    tonConveyorLevelerHomingTimeout(IN := FALSE);
    tonConveyorLevelerBrakeReleaseDelay(IN := FALSE);
    tonConveyorLevelerBrakeHoldDelay(IN := FALSE);

    conveyorLevelerFault := TRUE;
    conveyorLevelerFaultCode := 2;
    conveyorLevelerControlState := E_ConveyorLevelerState.FAULT;


ELSIF NOT conveyorLevelerDriveOk THEN

    conveyorLevelerState := 'DRIVE_NOT_OK';

    tonConveyorLevelerHomingTimeout(IN := FALSE);
    tonConveyorLevelerBrakeReleaseDelay(IN := FALSE);
    tonConveyorLevelerBrakeHoldDelay(IN := FALSE);

    conveyorLevelerFault := TRUE;
    conveyorLevelerFaultCode := 1;
    conveyorLevelerControlState := E_ConveyorLevelerState.FAULT;


ELSIF conveyorLevelerUpperSafetyLimit THEN

    conveyorLevelerState := 'UPPER_SAFE_LIMIT';

    tonConveyorLevelerHomingTimeout(IN := FALSE);
    tonConveyorLevelerBrakeReleaseDelay(IN := FALSE);
    tonConveyorLevelerBrakeHoldDelay(IN := FALSE);

    conveyorLevelerFault := TRUE;
    conveyorLevelerFaultCode := 4;
    conveyorLevelerControlState := E_ConveyorLevelerState.FAULT;


ELSIF conveyorLevelerLowerSafetyLimit THEN

    conveyorLevelerState := 'LOWER_SAFE_LIMIT';

    tonConveyorLevelerHomingTimeout(IN := FALSE);
    tonConveyorLevelerBrakeReleaseDelay(IN := FALSE);
    tonConveyorLevelerBrakeHoldDelay(IN := FALSE);

    conveyorLevelerFault := TRUE;
    conveyorLevelerFaultCode := 5;
    conveyorLevelerControlState := E_ConveyorLevelerState.FAULT;


ELSIF NOT systemRunEnable THEN

    // EN: Master stop disables movement without generating an axis fault.
    conveyorLevelerState := 'SYSTEM_DISABLED';

    conveyorLevelerSignedSpeedRefMmps := 0.0;

    tonConveyorLevelerHomingTimeout(IN := FALSE);
    tonConveyorLevelerBrakeReleaseDelay(IN := FALSE);
    tonConveyorLevelerBrakeHoldDelay(IN := FALSE);

    IF conveyorLevelerControlState <> E_ConveyorLevelerState.FAULT THEN
        conveyorLevelerControlState := E_ConveyorLevelerState.STOP;
    END_IF


ELSE

    //==============================================================
    // 9) Mode selection
    //==============================================================
    // EN: Homing has priority over manual and automatic leveling.
    IF rConveyorLevelerHome AND NOT conveyorLevelerFault THEN
        conveyorLevelerControlState := E_ConveyorLevelerState.HOME_FAST_SEARCH;
    END_IF;


    //==============================================================
    // 10) Conveyor leveler state machine
    //==============================================================
    CASE conveyorLevelerControlState OF

        E_ConveyorLevelerState.STOP: // STOP
            conveyorLevelerState := 'STOP';

            tonConveyorLevelerHomingTimeout(IN := FALSE);

            IF conveyorLevelerUpCmd OR conveyorLevelerDownCmd THEN

                conveyorLevelerControlState := E_ConveyorLevelerState.MANUAL;

            ELSIF conveyorLevelerAutoCmd THEN

                conveyorLevelerControlState := E_ConveyorLevelerState.AUTO_LEVELING;

            END_IF


        E_ConveyorLevelerState.HOME_FAST_SEARCH: // HOME_FAST_SEARCH
            conveyorLevelerState := 'HOME_FAST';

            conveyorLevelerHomed := FALSE;
            conveyorLevelerInPosition := FALSE;

            tonConveyorLevelerHomingTimeout(
                IN := TRUE,
                PT := machineConfig.conveyorLevelerHomingTimeout
            );

            IF tonConveyorLevelerHomingTimeout.Q THEN

                conveyorLevelerSignedSpeedRefMmps := 0.0;

                tonConveyorLevelerHomingTimeout(IN := FALSE);

                conveyorLevelerFault := TRUE;
                conveyorLevelerFaultCode := 3;

                conveyorLevelerState := 'HOME_TIMEOUT';
                conveyorLevelerControlState := E_ConveyorLevelerState.FAULT;


            ELSIF conveyorLevelerHomeLimitReached THEN

                // EN: Lower home sensor found. Stop and start slow exit.
                conveyorLevelerSignedSpeedRefMmps := 0.0;

                conveyorLevelerControlState := E_ConveyorLevelerState.HOME_SLOW_EXIT_SENSOR;


            ELSE

                IF conveyorLevelerHomeMoveAllowed THEN

                    // EN: Fast search moves down to find the lower home sensor.
                    conveyorLevelerSignedSpeedRefMmps :=
                        -ABS(machineConfig.conveyorLevelerHomingSpeedMmps);

                ELSE

                    conveyorLevelerSignedSpeedRefMmps := 0.0;

                END_IF

            END_IF


        E_ConveyorLevelerState.HOME_SLOW_EXIT_SENSOR: // HOME_SLOW_EXIT_SENSOR
            conveyorLevelerState := 'HOME_SLOW_EXIT';

            tonConveyorLevelerHomingTimeout(
                IN := TRUE,
                PT := machineConfig.conveyorLevelerHomingTimeout
            );

            IF tonConveyorLevelerHomingTimeout.Q THEN

                conveyorLevelerSignedSpeedRefMmps := 0.0;

                tonConveyorLevelerHomingTimeout(IN := FALSE);

                conveyorLevelerFault := TRUE;
                conveyorLevelerFaultCode := 3;

                conveyorLevelerState := 'HOME_TIMEOUT';
                conveyorLevelerControlState := E_ConveyorLevelerState.FAULT;


            ELSIF conveyorLevelerHomeLimitFallingEdge THEN

                // EN: Lower home sensor falling edge found.
                //     Stop before setting encoder.
                conveyorLevelerSignedSpeedRefMmps := 0.0;

                tonConveyorLevelerHomingTimeout(IN := FALSE);

                conveyorLevelerControlState := E_ConveyorLevelerState.HOME_SET_ENCODER;


            ELSE

                IF conveyorLevelerHomeMoveAllowed THEN

                    // EN: Slow exit moves up until leaving the lower home sensor.
                    conveyorLevelerSignedSpeedRefMmps :=
                        ABS(machineConfig.conveyorLevelerMinMoveSpeedMmps);

                ELSE

                    conveyorLevelerSignedSpeedRefMmps := 0.0;

                END_IF

            END_IF


        E_ConveyorLevelerState.HOME_SET_ENCODER: // HOME_SET_ENCODER
            conveyorLevelerState := 'HOME_SET_ENCODER';

            conveyorLevelerSignedSpeedRefMmps := 0.0;

            tonConveyorLevelerHomingTimeout(IN := FALSE);

            // EN: Set encoder only after leaving the home sensor edge.
            conveyorLevelerSetEncoderPositionTrigger := TRUE;
            conveyorLevelerSetEncoderPositionMm :=
                machineConfig.conveyorLevelerMinPositionMm;

            conveyorLevelerHomed := TRUE;
            conveyorLevelerFault := FALSE;
            conveyorLevelerFaultCode := 0;

            IF conveyorLevelerAutoCmd THEN
                conveyorLevelerControlState := E_ConveyorLevelerState.AUTO_LEVELING;
            ELSE
                conveyorLevelerControlState := E_ConveyorLevelerState.STOP;
            END_IF


        E_ConveyorLevelerState.MANUAL: // MANUAL
            conveyorLevelerState := 'MANUAL';

            tonConveyorLevelerHomingTimeout(IN := FALSE);

            IF conveyorLevelerUpCmd AND conveyorLevelerDownCmd THEN

                conveyorLevelerSignedSpeedRefMmps := 0.0;


            ELSIF conveyorLevelerUpCmd THEN

                IF conveyorLevelerUpAllowed THEN

                    conveyorLevelerSignedSpeedRefMmps :=
                        ABS(machineConfig.conveyorLevelerManualSpeedMmps);

                ELSE

                    conveyorLevelerSignedSpeedRefMmps := 0.0;

                END_IF


            ELSIF conveyorLevelerDownCmd THEN

                IF conveyorLevelerDownAllowed THEN

                    conveyorLevelerSignedSpeedRefMmps :=
                        -ABS(machineConfig.conveyorLevelerManualSpeedMmps);

                ELSE

                    conveyorLevelerSignedSpeedRefMmps := 0.0;

                END_IF


            ELSE

                conveyorLevelerSignedSpeedRefMmps := 0.0;

                IF conveyorLevelerAutoCmd THEN

                    conveyorLevelerControlState := E_ConveyorLevelerState.AUTO_LEVELING;

                ELSE

                    conveyorLevelerControlState := E_ConveyorLevelerState.STOP;

                END_IF

            END_IF


        E_ConveyorLevelerState.AUTO_LEVELING: // AUTO_LEVELING
            conveyorLevelerState := 'AUTO_LEVELING';

            tonConveyorLevelerHomingTimeout(IN := FALSE);

            IF NOT conveyorLevelerAutoCmd THEN

                conveyorLevelerSignedSpeedRefMmps := 0.0;
                conveyorLevelerControlState := E_ConveyorLevelerState.STOP;


            ELSIF NOT conveyorLevelerHomed THEN

                // EN: Automatic leveling is blocked before homing.
                conveyorLevelerSignedSpeedRefMmps := 0.0;
                conveyorLevelerState := 'AUTO_NO_HOME';


            ELSIF conveyorLevelerInPosition THEN

                conveyorLevelerSignedSpeedRefMmps := 0.0;


            ELSE

                // EN: Simple proportional position control.
                conveyorLevelerRawSpeedRefMmps :=
                    conveyorLevelerPositionErrorMm *
                    machineConfig.conveyorLevelerPositionKp;

                conveyorLevelerRawSpeedRefMmps :=
                    LIMIT(
                        -ABS(machineConfig.conveyorLevelerAutoMaxSpeedMmps),
                        conveyorLevelerRawSpeedRefMmps,
                        ABS(machineConfig.conveyorLevelerAutoMaxSpeedMmps)
                    );

                // EN: Apply minimum movement speed to overcome friction.
                IF ABS(conveyorLevelerRawSpeedRefMmps) <
                   ABS(machineConfig.conveyorLevelerMinMoveSpeedMmps) THEN

                    IF conveyorLevelerPositionErrorMm > 0.0 THEN

                        conveyorLevelerRawSpeedRefMmps :=
                            ABS(machineConfig.conveyorLevelerMinMoveSpeedMmps);

                    ELSE

                        conveyorLevelerRawSpeedRefMmps :=
                            -ABS(machineConfig.conveyorLevelerMinMoveSpeedMmps);

                    END_IF

                END_IF

                // EN: Apply limit protection according to movement direction.
                IF (conveyorLevelerRawSpeedRefMmps > 0.0) AND conveyorLevelerUpAllowed THEN

                    conveyorLevelerSignedSpeedRefMmps := conveyorLevelerRawSpeedRefMmps;

                ELSIF (conveyorLevelerRawSpeedRefMmps < 0.0) AND conveyorLevelerDownAllowed THEN

                    conveyorLevelerSignedSpeedRefMmps := conveyorLevelerRawSpeedRefMmps;

                ELSE

                    conveyorLevelerSignedSpeedRefMmps := 0.0;

                END_IF

            END_IF


        E_ConveyorLevelerState.FAULT: // FAULT
            conveyorLevelerState := 'FAULT';

            conveyorLevelerSignedSpeedRefMmps := 0.0;

            tonConveyorLevelerHomingTimeout(IN := FALSE);

            IF resetCmd AND
               safetyCircuitOk AND
               conveyorLevelerDriveOk AND
               NOT conveyorLevelerUpperSafetyLimit AND
               NOT conveyorLevelerLowerSafetyLimit THEN

                conveyorLevelerFault := FALSE;
                conveyorLevelerFaultCode := 0;
                conveyorLevelerControlState := E_ConveyorLevelerState.STOP;

            END_IF


    ELSE

        conveyorLevelerControlState := E_ConveyorLevelerState.STOP;

    END_CASE;

END_IF;


//==============================================================
// 11) Encoder set pulse
//==============================================================
// EN: Extend encoder set command to ensure the encoder block sees it.
tpConveyorLevelerSetEncoderPosition(
    IN := conveyorLevelerSetEncoderPositionTrigger,
    PT := machineConfig.conveyorLevelerSetEncoderPulseTime
);

conveyorLevelerSetEncoderPosition := tpConveyorLevelerSetEncoderPosition.Q;


//==============================================================
// 12) Brake release control
//==============================================================
// EN: A movement request keeps the magnetic brake released.
//     After movement stops, the brake remains released for a hold time.
conveyorLevelerMoveRequest :=
    systemRunEnable AND
    safetyCircuitOk AND
    conveyorLevelerDriveOk AND
    NOT conveyorLevelerFault AND
    (ABS(conveyorLevelerSignedSpeedRefMmps) >= machineConfig.conveyorLevelerRunMinSpeedMmps);


IF conveyorLevelerMoveRequest THEN

    conveyorLevelerBrakeReleaseRequest := TRUE;

    tonConveyorLevelerBrakeHoldDelay(IN := FALSE);

ELSE

    IF conveyorLevelerBrakeRelease THEN

        tonConveyorLevelerBrakeHoldDelay(
            IN := TRUE,
            PT := machineConfig.conveyorLevelerBrakeHoldTime
        );

        conveyorLevelerBrakeReleaseRequest :=
            NOT tonConveyorLevelerBrakeHoldDelay.Q;

    ELSE

        tonConveyorLevelerBrakeHoldDelay(IN := FALSE);
        conveyorLevelerBrakeReleaseRequest := FALSE;

    END_IF

END_IF;


conveyorLevelerBrakeRelease :=
    systemRunEnable AND
    safetyCircuitOk AND
    conveyorLevelerDriveOk AND
    NOT conveyorLevelerFault AND
    conveyorLevelerBrakeReleaseRequest;


//==============================================================
// 13) Brake release delay before motor movement
//==============================================================
// EN: The motor can run only after brake release delay.
tonConveyorLevelerBrakeReleaseDelay(
    IN := conveyorLevelerMoveRequest AND conveyorLevelerBrakeRelease,
    PT := machineConfig.conveyorLevelerBrakeReleaseDelay
);


//==============================================================
// 14) Conveyor leveler direction and speed outputs
//==============================================================
// EN: Convert signed internal speed command into direction outputs
//     and positive speed reference.
IF conveyorLevelerMoveRequest AND
   conveyorLevelerBrakeRelease AND
   tonConveyorLevelerBrakeReleaseDelay.Q THEN

    conveyorLevelerSpeedRefMmps :=
        ABS(conveyorLevelerSignedSpeedRefMmps);

    conveyorLevelerRunUp :=
        conveyorLevelerSignedSpeedRefMmps > 0.0;

    conveyorLevelerRunDown :=
        conveyorLevelerSignedSpeedRefMmps < 0.0;

ELSE

    conveyorLevelerSpeedRefMmps := 0.0;

    conveyorLevelerRunUp := FALSE;
    conveyorLevelerRunDown := FALSE;

END_IF;
END_METHOD

//==============================================================
// SIMPLE STACKER — SPEED REFERENCE GENERATOR
// EN: Generates synchronized and sheet-stack separation speed references [m/min].
//==============================================================
METHOD _ConveyorSpeedControl
VAR
packageGapReady                   : BOOL;
    validCycleTimeS                   : REAL;

    sheetConveyorsSpeedUpReferenceMPM : REAL;

    sheetConveyor1BaseSpeedMPM        : REAL;
    sheetConveyor2BaseSpeedMPM        : REAL;
    sheetConveyor3BaseSpeedMPM        : REAL;
END_VAR


//==============================================================
// 1) Default event pulses
//==============================================================
sheetStackSeparationStarted         := FALSE;
sheetStackSeparationFinished        := FALSE;

sheetConveyor2SeparationStarted     := FALSE;
sheetConveyor2SeparationFinished    := FALSE;

sheetConveyor3SeparationStarted     := FALSE;
sheetConveyor3SeparationFinished    := FALSE;


//==============================================================
// 2) Enable and scan time
//==============================================================
speedControlEnabled :=
    sheetConveyor1Run AND
    sheetConveyor2Run AND
    sheetConveyor3Run AND
    safetyCircuitOk;

rampReset := NOT speedControlEnabled;


// EN: Read PLC scan time using OSCAT CYCLE_TIME.
instCycleTime(
    RST := resetCmd
);


// EN: Convert last cycle time from TIME/ms to seconds.
scanTimeMs := TIME_TO_REAL(instCycleTime.ct_last);

validCycleTimeS :=
    LIMIT(
        0.001,
        scanTimeMs / 1000.0,
        20.0
    );

scanTimeS := validCycleTimeS;



//==============================================================
// 4) Calculate normal stacker speed
//==============================================================
IF speedControlEnabled THEN

    normalStackerSpeedMPM :=
        LIMIT(
            machineConfig.minimumSpeedMPM,
            MAX(0.0, lineSpeedMPM) *
                MAX(0.0, machineConfig.stackerSpeedRatio),
            machineConfig.maximumSpeedMPM
        );

ELSE

    normalStackerSpeedMPM := 0.0;

END_IF;


//==============================================================
// 6) Calculate normal speed for each conveyor
//==============================================================
sheetConveyor1NormalSpeedMPM :=
    normalStackerSpeedMPM *
    MAX(0.0, machineConfig.sheetConveyor1SpeedTrim);

sheetConveyor2NormalSpeedMPM :=
    normalStackerSpeedMPM *
    MAX(0.0, machineConfig.sheetConveyor2SpeedTrim);

sheetConveyor3NormalSpeedMPM :=
    normalStackerSpeedMPM *
    MAX(0.0, machineConfig.sheetConveyor3SpeedTrim);


//==============================================================
// 6.1) Sheet conveyors speed-up reference
//==============================================================
// EN: Speed-up is added directly to conveyors 1/2/3 references.
//     It can work even when line speed is zero, as long as the
//     conveyor group is enabled.
IF speedControlEnabled AND sheetConveyorsSpeedUpCmd THEN

    sheetConveyorsSpeedUpReferenceMPM :=
        MAX(0.0, machineConfig.sheetConveyorsSpeedUpMPM);

ELSE

    sheetConveyorsSpeedUpReferenceMPM := 0.0;

END_IF;


//==============================================================
// 6.2) Base speed references including speed-up
//==============================================================
// EN: Base speed is the synchronized conveyor speed plus operator speed-up.
//     Separation tracking must use this base speed as reference.
sheetConveyor1BaseSpeedMPM :=
    sheetConveyor1NormalSpeedMPM + sheetConveyorsSpeedUpReferenceMPM;

sheetConveyor2BaseSpeedMPM :=
    sheetConveyor2NormalSpeedMPM + sheetConveyorsSpeedUpReferenceMPM;

sheetConveyor3BaseSpeedMPM :=
    sheetConveyor3NormalSpeedMPM + sheetConveyorsSpeedUpReferenceMPM;


//==============================================================
// 7) Calculate separation high speed
//==============================================================
// EN: Gap speed also receives the same speed-up reference.
//     This preserves the real gap differential while allowing operator boost.
sheetConveyor2GapSpeedMPM :=
    (sheetConveyor2NormalSpeedMPM * MAX(0.0, machineConfig.packageGapSpeedRatio)) +
    machineConfig.packageGapSpeedOffsetMPM +
    sheetConveyorsSpeedUpReferenceMPM;

sheetConveyor3GapSpeedMPM :=
    (sheetConveyor3NormalSpeedMPM * MAX(0.0, machineConfig.packageGapSpeedRatio)) +
    machineConfig.packageGapSpeedOffsetMPM +
    sheetConveyorsSpeedUpReferenceMPM;


//==============================================================
// 8) Calculate separation tracking target distances
//==============================================================
// EN: Separation tracking target is based on each conveyor length.
sheetConveyor2TargetDistanceM :=
    MAX(0.0, machineConfig.sheetConveyor2LengthM);

sheetConveyor3TargetDistanceM :=
    MAX(0.0, machineConfig.sheetConveyor3LengthM);


//==============================================================
// 9) Check separation ready conditions
//==============================================================
// EN: Compare gap speed against base speed, not normal speed.
//     Otherwise operator speed-up would be incorrectly counted as gap opening.
packageGapReady :=
    speedControlEnabled AND
    (sheetConveyor2TargetDistanceM > 0.0) AND
    (sheetConveyor3TargetDistanceM > 0.0) AND
    ((sheetConveyor2GapSpeedMPM - sheetConveyor2BaseSpeedMPM) >= machineConfig.minimumOpeningSpeedMPM) AND
    ((sheetConveyor3GapSpeedMPM - sheetConveyor3BaseSpeedMPM) >= machineConfig.minimumOpeningSpeedMPM);

sheetStackSeparationReady := packageGapReady;


//==============================================================
// 9) Sheet stack separation state machine
//==============================================================
IF NOT speedControlEnabled THEN

    sheetStackSeparationState      := 'DISABLED';
    sheetStackSeparationStateCode  := -1;

    packageSeparationState         := E_PackageSeparationState.NORMAL;

    sheetStackSeparationActive     := FALSE;
    sheetStackBrakeActive          := FALSE;
    brakeValve                     := FALSE;

    sheetConveyor2SeparationActive := FALSE;
    sheetConveyor3SeparationActive := FALSE;

    sheetConveyor2HighSpeedActive  := FALSE;
    sheetConveyor3HighSpeedActive  := FALSE;

    sheetConveyor2OpeningDistanceM := 0.0;
    sheetConveyor3OpeningDistanceM := 0.0;

    sheetConveyor1TargetSpeedMPM   := 0.0;
    sheetConveyor2TargetSpeedMPM   := 0.0;
    sheetConveyor3TargetSpeedMPM   := 0.0;


ELSE

    CASE packageSeparationState OF

        E_PackageSeparationState.NORMAL: // NORMAL
            sheetStackSeparationState     := 'NORMAL';
            sheetStackSeparationStateCode := 0;

            sheetStackSeparationActive    := FALSE;
            sheetStackBrakeActive         := FALSE;
            brakeValve                    := FALSE;

            sheetConveyor2SeparationActive := FALSE;
            sheetConveyor3SeparationActive := FALSE;

            sheetConveyor2HighSpeedActive  := FALSE;
            sheetConveyor3HighSpeedActive  := FALSE;

            sheetConveyor2OpeningDistanceM := 0.0;
            sheetConveyor3OpeningDistanceM := 0.0;

            sheetConveyor1TargetSpeedMPM  := sheetConveyor1BaseSpeedMPM;
            sheetConveyor2TargetSpeedMPM  := sheetConveyor2BaseSpeedMPM;
            sheetConveyor3TargetSpeedMPM  := sheetConveyor3BaseSpeedMPM;

            IF rPackageComplete AND packageGapReady THEN
                packageSeparationState := E_PackageSeparationState.START_SEPARATION;
            END_IF


        E_PackageSeparationState.START_SEPARATION: // START_SHEET_STACK_SEPARATION
            sheetStackSeparationState     := 'START_SEPARATION';
            sheetStackSeparationStateCode := 10;

            sheetStackSeparationActive    := TRUE;
            sheetStackSeparationStarted   := TRUE;

            sheetStackBrakeActive         := TRUE;
            brakeValve                    := TRUE;

            // EN: Conveyor 2 tracking starts immediately.
            sheetConveyor2SeparationStarted := TRUE;

            sheetConveyor2SeparationActive  := TRUE;
            sheetConveyor3SeparationActive  := FALSE;

            // EN: Conveyor 2 and 3 accelerate together from the beginning.
            sheetConveyor2HighSpeedActive   := TRUE;
            sheetConveyor3HighSpeedActive   := TRUE;

            sheetConveyor2OpeningDistanceM  := 0.0;
            sheetConveyor3OpeningDistanceM  := 0.0;

            sheetConveyor1TargetSpeedMPM    := sheetConveyor1BaseSpeedMPM;
            sheetConveyor2TargetSpeedMPM    := sheetConveyor2GapSpeedMPM;
            sheetConveyor3TargetSpeedMPM    := sheetConveyor3GapSpeedMPM;

            packageSeparationState := E_PackageSeparationState.CONVEYOR_2_TRACKING;


        E_PackageSeparationState.CONVEYOR_2_TRACKING: // SHEET_CONVEYOR_2_SEPARATION_TRACKING
            sheetStackSeparationState     := 'CONV2_TRACKING';
            sheetStackSeparationStateCode := 20;

            sheetStackSeparationActive    := TRUE;

            sheetStackBrakeActive         := TRUE;
            brakeValve                    := TRUE;

            sheetConveyor2SeparationActive := TRUE;
            sheetConveyor3SeparationActive := FALSE;

            sheetConveyor2HighSpeedActive  := TRUE;
            sheetConveyor3HighSpeedActive  := TRUE;

            sheetConveyor1TargetSpeedMPM  := sheetConveyor1BaseSpeedMPM;
            sheetConveyor2TargetSpeedMPM  := sheetConveyor2GapSpeedMPM;
            sheetConveyor3TargetSpeedMPM  := sheetConveyor3GapSpeedMPM;

            IF sheetConveyor2OpeningDistanceM >= sheetConveyor2TargetDistanceM THEN

                // EN: Conveyor 2 tracking finished. Conveyor 2 returns to base speed.
                sheetConveyor2SeparationFinished := TRUE;

                sheetConveyor2SeparationActive   := FALSE;
                sheetConveyor2HighSpeedActive    := FALSE;

                sheetStackBrakeActive            := FALSE;
                brakeValve                       := FALSE;

                sheetConveyor2TargetSpeedMPM     := sheetConveyor2BaseSpeedMPM;

                // EN: Conveyor 3 tracking starts after conveyor 2 returns to sync.
                sheetConveyor3SeparationStarted := TRUE;
                sheetConveyor3OpeningDistanceM  := 0.0;

                packageSeparationState := E_PackageSeparationState.CONVEYOR_3_TRACKING;

            END_IF


        E_PackageSeparationState.CONVEYOR_3_TRACKING: // SHEET_CONVEYOR_3_SEPARATION_TRACKING
            sheetStackSeparationState     := 'CONV3_TRACKING';
            sheetStackSeparationStateCode := 30;

            sheetStackSeparationActive    := TRUE;

            sheetStackBrakeActive         := FALSE;
            brakeValve                    := FALSE;

            sheetConveyor2SeparationActive := FALSE;
            sheetConveyor3SeparationActive := TRUE;

            sheetConveyor2HighSpeedActive  := FALSE;
            sheetConveyor3HighSpeedActive  := TRUE;

            sheetConveyor1TargetSpeedMPM  := sheetConveyor1BaseSpeedMPM;
            sheetConveyor2TargetSpeedMPM  := sheetConveyor2BaseSpeedMPM;
            sheetConveyor3TargetSpeedMPM  := sheetConveyor3GapSpeedMPM;

            IF sheetConveyor3OpeningDistanceM >= sheetConveyor3TargetDistanceM THEN

                // EN: Conveyor 3 returns to base synchronized speed.
                sheetConveyor3TargetSpeedMPM := sheetConveyor3BaseSpeedMPM;

                packageSeparationState := E_PackageSeparationState.FINISH_SEPARATION;

            END_IF


        E_PackageSeparationState.FINISH_SEPARATION: // FINISH_SHEET_STACK_SEPARATION
            sheetStackSeparationState     := 'FINISH_SEPARATION';
            sheetStackSeparationStateCode := 40;

            sheetStackSeparationActive    := FALSE;
            sheetStackSeparationFinished  := TRUE;

            sheetStackBrakeActive         := FALSE;
            brakeValve                    := FALSE;

            sheetConveyor2SeparationActive  := FALSE;
            sheetConveyor3SeparationActive  := FALSE;

            sheetConveyor2HighSpeedActive   := FALSE;
            sheetConveyor3HighSpeedActive   := FALSE;

            sheetConveyor3SeparationFinished := TRUE;

            sheetConveyor1TargetSpeedMPM  := sheetConveyor1BaseSpeedMPM;
            sheetConveyor2TargetSpeedMPM  := sheetConveyor2BaseSpeedMPM;
            sheetConveyor3TargetSpeedMPM  := sheetConveyor3BaseSpeedMPM;

            packageSeparationState := E_PackageSeparationState.NORMAL;


    ELSE

        packageSeparationState := E_PackageSeparationState.NORMAL;

    END_CASE;

END_IF;


//==============================================================
// 10) Limit speed targets
//==============================================================
sheetConveyor1TargetSpeedMPM := LIMIT(
    machineConfig.minimumSpeedMPM,
    sheetConveyor1TargetSpeedMPM,
    machineConfig.maximumSpeedMPM
);

sheetConveyor2TargetSpeedMPM := LIMIT(
    machineConfig.minimumSpeedMPM,
    sheetConveyor2TargetSpeedMPM,
    machineConfig.maximumSpeedMPM
);

sheetConveyor3TargetSpeedMPM := LIMIT(
    machineConfig.minimumSpeedMPM,
    sheetConveyor3TargetSpeedMPM,
    machineConfig.maximumSpeedMPM
);


//==============================================================
// 12) Ramp sheet conveyor 1 speed reference
//==============================================================
instRampSheetConveyor1(
    X          := sheetConveyor1TargetSpeedMPM,
    A_UP       := MAX(0.0, machineConfig.rampAccelerationUpMPMps2),
    A_DN       := -MAX(0.0, machineConfig.rampAccelerationDownMPMps2),
    VU_MAX     := MAX(0.0, machineConfig.rampVelocityUpMaxMPMps),
    VD_MAX     := -MAX(0.0, machineConfig.rampVelocityDownMaxMPMps),
    LIMIT_HIGH := machineConfig.maximumSpeedMPM,
    LIMIT_LOW  := machineConfig.minimumSpeedMPM,
    RST        := rampReset,
    Y          => sheetConveyor1SpeedRefMPM
);


//==============================================================
// 13) Ramp sheet conveyor 2 speed reference
//==============================================================
instRampSheetConveyor2(
    X          := sheetConveyor2TargetSpeedMPM,
    A_UP       := MAX(0.0, machineConfig.rampAccelerationUpMPMps2),
    A_DN       := -MAX(0.0, machineConfig.rampAccelerationDownMPMps2),
    VU_MAX     := MAX(0.0, machineConfig.rampVelocityUpMaxMPMps),
    VD_MAX     := -MAX(0.0, machineConfig.rampVelocityDownMaxMPMps),
    LIMIT_HIGH := machineConfig.maximumSpeedMPM,
    LIMIT_LOW  := machineConfig.minimumSpeedMPM,
    RST        := rampReset,
    Y          => sheetConveyor2SpeedRefMPM
);


//==============================================================
// 14) Ramp sheet conveyor 3 speed reference
//==============================================================
instRampSheetConveyor3(
    X          := sheetConveyor3TargetSpeedMPM,
    A_UP       := MAX(0.0, machineConfig.rampAccelerationUpMPMps2),
    A_DN       := -MAX(0.0, machineConfig.rampAccelerationDownMPMps2),
    VU_MAX     := MAX(0.0, machineConfig.rampVelocityUpMaxMPMps),
    VD_MAX     := -MAX(0.0, machineConfig.rampVelocityDownMaxMPMps),
    LIMIT_HIGH := machineConfig.maximumSpeedMPM,
    LIMIT_LOW  := machineConfig.minimumSpeedMPM,
    RST        := rampReset,
    Y          => sheetConveyor3SpeedRefMPM
);


//==============================================================
// 16) Calculate real separation tracking speed using ramped references
//==============================================================
// EN: Only the real speed differential above the base speed moves the
//     separation point through the conveyors.
//     Operator speed-up is already included in base speed, so it is not
//     counted as gap opening.
sheetConveyor2OpeningSpeedMPM :=
    MAX(0.0, sheetConveyor2SpeedRefMPM - sheetConveyor2BaseSpeedMPM);

sheetConveyor3OpeningSpeedMPM :=
    MAX(0.0, sheetConveyor3SpeedRefMPM - sheetConveyor3BaseSpeedMPM);


//==============================================================
// 17) Integrate real separation tracking distance
//==============================================================
IF speedControlEnabled THEN

    IF packageSeparationState = E_PackageSeparationState.CONVEYOR_2_TRACKING THEN

        IF sheetConveyor2OpeningSpeedMPM >= machineConfig.minimumOpeningSpeedMPM THEN

            sheetConveyor2OpeningDistanceM :=
                sheetConveyor2OpeningDistanceM +
                (sheetConveyor2OpeningSpeedMPM / 60.0) * scanTimeS;

        END_IF

    ELSIF packageSeparationState = E_PackageSeparationState.CONVEYOR_3_TRACKING THEN

        IF sheetConveyor3OpeningSpeedMPM >= machineConfig.minimumOpeningSpeedMPM THEN

            sheetConveyor3OpeningDistanceM :=
                sheetConveyor3OpeningDistanceM +
                (sheetConveyor3OpeningSpeedMPM / 60.0) * scanTimeS;

        END_IF

    END_IF

END_IF;


//==============================================================
// 18) Publish tracking distances to outputs
//==============================================================
sheetConveyor2TrackingDistanceM := sheetConveyor2OpeningDistanceM;
sheetConveyor3TrackingDistanceM := sheetConveyor3OpeningDistanceM;
END_METHOD

//==============================================================
// SIMPLE STACKER — HMI STATUS
// EN: Maps internal status, outputs, positions and diagnostics
//     to the HMI status structure.
//==============================================================
METHOD _HmiStatus



//==============================================================
// 1) System general status
//==============================================================
hmiStatus.systemRunEnable :=
    systemRunEnable;

hmiStatus.safetyCircuitOk :=
    safetyCircuitOk;

hmiStatus.faultActive :=
    faultActive OR
    backstopFault OR
    conveyorLevelerFault OR
    sheetStackDischargeFault OR
    sheetStackDischargeConveyorFault;

hmiStatus.deviceState :=
    deviceState;


//==============================================================
// 2) Sheet conveyor group status
//==============================================================
hmiStatus.synchronizedConveyorsRunning :=
    synchronizedConveyorsRunning;

hmiStatus.sheetConveyor1Run :=
    sheetConveyor1Run;

hmiStatus.sheetConveyor2Run :=
    sheetConveyor2Run;

hmiStatus.sheetConveyor3Run :=
    sheetConveyor3Run;

hmiStatus.sheetConveyor1SpeedRefMPM :=
    sheetConveyor1SpeedRefMPM;

hmiStatus.sheetConveyor2SpeedRefMPM :=
    sheetConveyor2SpeedRefMPM;

hmiStatus.sheetConveyor3SpeedRefMPM :=
    sheetConveyor3SpeedRefMPM;

CASE syncConveyorsState OF
    E_SyncConveyorsState.IDLE:
        hmiStatus.syncConveyorsState := 0;

    E_SyncConveyorsState.RUN:
        hmiStatus.syncConveyorsState := 1;

    E_SyncConveyorsState.FAULT:
        hmiStatus.syncConveyorsState := 10;

ELSE
    hmiStatus.syncConveyorsState := 0;
END_CASE;


//==============================================================
// 3) Sheet stack separation status
//==============================================================
hmiStatus.sheetStackSeparationReady :=
    sheetStackSeparationReady;

hmiStatus.sheetStackSeparationActive :=
    sheetStackSeparationActive;

hmiStatus.sheetStackBrakeActive :=
    sheetStackBrakeActive;


//==============================================================
// 4) Sheet stack discharge sequence status
//==============================================================
hmiStatus.sheetStackDischargeState :=
    sheetStackDischargeState;

hmiStatus.sheetStackDischargeStateCode :=
    sheetStackDischargeStateCode;

hmiStatus.sheetStackDischargePending :=
    sheetStackDischargePending;

hmiStatus.sheetStackDischargeActive :=
    sheetStackDischargeActive;

hmiStatus.sheetStackDischargeStarted :=
    sheetStackDischargeStarted;

hmiStatus.sheetStackDischargeFinished :=
    sheetStackDischargeFinished;

hmiStatus.sheetStackDischargeFault :=
    sheetStackDischargeFault;

hmiStatus.sheetStackDischargeFaultCode :=
    sheetStackDischargeFaultCode;

hmiStatus.sheetStackDischargeLastCycleOk :=
    sheetStackDischargeLastCycleOk;

hmiStatus.sheetStackDischargeLastResultCode :=
    sheetStackDischargeLastResultCode;

hmiStatus.sheetStackDischargeLastFaultStepCode :=
    sheetStackDischargeLastFaultStepCode;

hmiStatus.sheetStackDischargeLastFaultCode :=
    sheetStackDischargeLastFaultCode;


//==============================================================
// 5) Sheet stack discharge conveyor status
//==============================================================
hmiStatus.sheetStackDischargeConveyorState :=
    sheetStackDischargeConveyorState;

hmiStatus.sheetStackDischargeConveyorRun :=
    sheetStackDischargeConveyorRun;

hmiStatus.sheetStackDischargeConveyorSpeedRefMPM :=
    sheetStackDischargeConveyorSpeedRefMPM;

hmiStatus.sheetStackDischargeConveyorFault :=
    sheetStackDischargeConveyorFault;

hmiStatus.sheetStackDischargeConveyorFaultCode :=
    sheetStackDischargeConveyorFaultCode;


//==============================================================
// 6) Backstop status
//==============================================================
hmiStatus.backstopState :=
    backstopState;

hmiStatus.backstopHomed :=
    backstopHomed;

hmiStatus.backstopHomeRunning :=
    backstopHomeRunning;

hmiStatus.backstopInPosition :=
    backstopInPosition;

hmiStatus.backstopPositionMm :=
    backstopPositionMm;

hmiStatus.backstopTargetPositionMm :=
    backstopTargetPositionMm;

hmiStatus.backstopPositionErrorMm :=
    backstopPositionErrorMm;

hmiStatus.backstopRunFw :=
    backstopRunFw;

hmiStatus.backstopRunRev :=
    backstopRunRev;

hmiStatus.backstopSpeedRefMmps :=
    backstopSpeedRefMmps;

hmiStatus.backstopPlateUpSolenoid :=
    backstopPlateUpSolenoid;

hmiStatus.backstopSetEncoderPosition :=
    backstopSetEncoderPosition;

hmiStatus.backstopSetEncoderPositionMm :=
    backstopSetEncoderPositionMm;

hmiStatus.backstopManualInterventionActive :=
    backstopManualInterventionActive;

hmiStatus.backstopManualInterventionPositionMm :=
    backstopManualInterventionPositionMm;

hmiStatus.backstopFault :=
    backstopFault;

hmiStatus.backstopFaultCode :=
    backstopFaultCode;


//==============================================================
// 7) Conveyor leveler status
//==============================================================
hmiStatus.conveyorLevelerState :=
    conveyorLevelerState;

hmiStatus.conveyorLevelerHomed :=
    conveyorLevelerHomed;

hmiStatus.conveyorLevelerInPosition :=
    conveyorLevelerInPosition;

hmiStatus.conveyorLevelerPositionMm :=
    conveyorLevelerPositionMm;

hmiStatus.conveyorLevelerTargetPositionMm :=
    conveyorLevelerTargetPositionMm;

hmiStatus.conveyorLevelerPositionErrorMm :=
    conveyorLevelerPositionErrorMm;

hmiStatus.conveyorLevelerRunUp :=
    conveyorLevelerRunUp;

hmiStatus.conveyorLevelerRunDown :=
    conveyorLevelerRunDown;

hmiStatus.conveyorLevelerBrakeRelease :=
    conveyorLevelerBrakeRelease;

hmiStatus.conveyorLevelerSpeedRefMmps :=
    conveyorLevelerSpeedRefMmps;

hmiStatus.conveyorLevelerSetEncoderPosition :=
    conveyorLevelerSetEncoderPosition;

hmiStatus.conveyorLevelerSetEncoderPositionMm :=
    conveyorLevelerSetEncoderPositionMm;

hmiStatus.conveyorLevelerFault :=
    conveyorLevelerFault;

hmiStatus.conveyorLevelerFaultCode :=
    conveyorLevelerFaultCode;


//==============================================================
// 8) Process values
//==============================================================
hmiStatus.lineSpeedMPM :=
    lineSpeedMPM;

hmiStatus.sheetLengthMm :=
    sheetLengthMm;

hmiStatus.stackHeightMm :=
    stackHeightMm;


//==============================================================
// 9) Input / drive status mirror
//==============================================================
hmiStatus.sheetConveyor1DriveOk :=
    sheetConveyor1DriveOk;

hmiStatus.sheetConveyor2DriveOk :=
    sheetConveyor2DriveOk;

hmiStatus.sheetConveyor3DriveOk :=
    sheetConveyor3DriveOk;

hmiStatus.backstopDriveOk :=
    backstopDriveOk;

hmiStatus.conveyorLevelerDriveOk :=
    conveyorLevelerDriveOk;

hmiStatus.sheetStackDischargeConveyorDriveOk :=
    sheetStackDischargeConveyorDriveOk;
END_METHOD

METHOD _MachineAuxiliary
VAR_INPUT
END_VAR
(*



stopMachinePulse :=
    NOT safetyCircuitOk OR
    NOT sheetConveyor1DriveOk OR
    NOT sheetConveyor2DriveOk OR
    NOT sheetConveyor3DriveOk;
	NOT backstopDriveOk
	NOT conveyorLevelerDriveOk
*)
noCrushRollersUpDownValve := noCrushRollersDownCmd;

stackerRunning := systemRunEnable;


reset := resetCmd;
END_METHOD

//==============================================================
// SIMPLE STACKER — SHEET CONVEYOR GROUP CONTROL
// EN: Controls the synchronized sheet conveyor group.
//     Start/stop command latch is handled by _SystemControl().
//==============================================================
METHOD _SheetConveyorGroupControl

//==============================================================
// 1) Conditions
//==============================================================
// EN: Only synchronized sheet conveyor drives are considered here.
// PT: Apenas os inversores das esteiras sincronizadas são considerados aqui.
allSynchronizedDrivesOk :=
    sheetConveyor1DriveOk AND
    sheetConveyor2DriveOk AND
    sheetConveyor3DriveOk;


// EN: Synchronized conveyor group fault.
// PT: Falha do grupo de esteiras sincronizadas.
anyFault :=
    NOT safetyCircuitOk OR
    NOT allSynchronizedDrivesOk;

faultActive := anyFault;


//==============================================================
// 2) State machine
//==============================================================
CASE syncConveyorsState OF

    E_SyncConveyorsState.IDLE: // IDLE
        deviceState := 'IDLE';

        sheetConveyor1Run := FALSE;
        sheetConveyor2Run := FALSE;
        sheetConveyor3Run := FALSE;

        synchronizedConveyorsRunning := FALSE;

        // EN: The group starts only when the master system is enabled
        //     and no conveyor group fault is active.
        IF systemRunEnable AND NOT anyFault THEN

            syncConveyorsState := E_SyncConveyorsState.RUN;

        ELSIF systemRunEnable AND anyFault THEN

            syncConveyorsState := E_SyncConveyorsState.FAULT;

        END_IF


    E_SyncConveyorsState.RUN: // RUN
        deviceState := 'RUN';

        // EN: Outputs are also directly conditioned by systemRunEnable
        //     to avoid one-scan movement after a stop command.
        sheetConveyor1Run :=
            systemRunEnable AND
            safetyCircuitOk AND
            sheetConveyor1DriveOk;

        sheetConveyor2Run :=
            systemRunEnable AND
            safetyCircuitOk AND
            sheetConveyor2DriveOk;

        sheetConveyor3Run :=
            systemRunEnable AND
            safetyCircuitOk AND
            sheetConveyor3DriveOk;

        synchronizedConveyorsRunning :=
            sheetConveyor1Run AND
            sheetConveyor2Run AND
            sheetConveyor3Run;

        IF anyFault THEN

            syncConveyorsState := E_SyncConveyorsState.FAULT;

        ELSIF NOT systemRunEnable THEN

            syncConveyorsState := E_SyncConveyorsState.IDLE;

        END_IF


    E_SyncConveyorsState.FAULT: // FAULT
        deviceState := 'FAULT';

        sheetConveyor1Run := FALSE;
        sheetConveyor2Run := FALSE;
        sheetConveyor3Run := FALSE;

        synchronizedConveyorsRunning := FALSE;

        // EN: Fault state is released only by reset and with all faults cleared.
        //     If systemRunEnable is still TRUE after reset, the group can start
        //     again from IDLE on the next scan.
        IF resetCmd AND NOT anyFault THEN

            syncConveyorsState := E_SyncConveyorsState.IDLE;

        END_IF


ELSE

    syncConveyorsState := E_SyncConveyorsState.IDLE;

END_CASE;
END_METHOD

//==============================================================
// SIMPLE STACKER — SHEET STACK DISCHARGE CONTROL
// EN: Controls the sheet stack discharge sequence after the sheet
//     conveyor separation cycle is completed.
//
// State code
// 0  = IDLE
// 5  = WAIT_SEPARATION
// 10 = START_DISCHARGE_POSITIONING
// 20 = WAIT_BACKSTOP_POSITION
// 30 = RUN_DISCHARGE_CONVEYOR
// 40 = START_RETURN_POSITIONING
// 50 = WAIT_BACKSTOP_RETURN
// 60 = FINISH
// 90 = ABORT_TRANSIENT
//
// Last result code
// 0 = No cycle executed yet
// 1 = Last cycle completed successfully
// 2 = Last cycle completed with manual backstop skip
// 3 = Last cycle completed/aborted by timeout
// 4 = Last cycle aborted by fault
//
// Fault code
// 0  = No fault
// 1  = Safety circuit not OK
// 2  = Sheet conveyor drive not OK
// 3  = Discharge conveyor drive/control fault
// 4  = Backstop drive/control fault
// 5  = Conveyor leveler drive/control fault
// 6  = Stacker stopped during cycle
// 10 = Wait separation timeout
// 20 = Backstop positioning timeout
// 30 = Discharge conveyor did not start timeout
// 50 = Backstop return timeout
//==============================================================
METHOD _SheetStackDischargeControl
VAR
    abortCycle : BOOL;
END_VAR


//==============================================================
// 1) Default event pulses
//==============================================================
sheetStackDischargeStarted  := FALSE;
sheetStackDischargeFinished := FALSE;


//==============================================================
// 2) Default internal requests / overrides
//==============================================================
// EN: The sequence does not write the physical discharge conveyor outputs.
//     It only generates an internal request to the conveyor control method.
sheetStackDischargeConveyorRunRequest := FALSE;

backstopTargetOverrideActive := FALSE;
backstopTargetOverridePositionMm := 0.0;

conveyorLevelerTargetOverrideActive := FALSE;
conveyorLevelerTargetOverridePositionMm := 0.0;


//==============================================================
// 3) Fault condition
//==============================================================
// EN: Conveyor leveler feedback is not used for sequence progress,
//     but its drive/control fault still aborts the cycle.
sheetStackDischargeFaultCondition :=
    NOT safetyCircuitOk OR
    NOT sheetConveyor1DriveOk OR
    NOT sheetConveyor2DriveOk OR
    NOT sheetConveyor3DriveOk OR
    NOT sheetStackDischargeConveyorDriveOk OR
    sheetStackDischargeConveyorFault OR
    NOT backstopDriveOk OR
    backstopFault OR
    NOT conveyorLevelerDriveOk OR
    conveyorLevelerFault;


//==============================================================
// 4) Fault code priority
//==============================================================
IF NOT safetyCircuitOk THEN

    sheetStackDischargeFaultCode := 1;

ELSIF NOT sheetConveyor1DriveOk OR
      NOT sheetConveyor2DriveOk OR
      NOT sheetConveyor3DriveOk THEN

    sheetStackDischargeFaultCode := 2;

ELSIF NOT sheetStackDischargeConveyorDriveOk OR
      sheetStackDischargeConveyorFault THEN

    sheetStackDischargeFaultCode := 3;

ELSIF NOT backstopDriveOk OR
      backstopFault THEN

    sheetStackDischargeFaultCode := 4;

ELSIF NOT conveyorLevelerDriveOk OR
      conveyorLevelerFault THEN

    sheetStackDischargeFaultCode := 5;

ELSIF NOT synchronizedConveyorsRunning THEN

    sheetStackDischargeFaultCode := 6;

END_IF;


//==============================================================
// 5) Optional reset of current sequence fault display
//==============================================================
// EN: Reset clears the current sequence fault flag,
//     but does not erase last cycle diagnostic codes.
IF resetCmd AND (sheetStackDischargeControlState = E_SheetStackDischargeState.IDLE) THEN

    sheetStackDischargeFault := FALSE;
    sheetStackDischargeFaultCode := 0;

END_IF;


//==============================================================
// 6) Arm discharge sequence from packageCompleteCmd
//==============================================================
// EN: packageCompleteCmd is ignored if stacker is not running or if
//     any relevant drive/safety fault is active.
IF rPackageCompleteDischarge AND
   synchronizedConveyorsRunning AND
   NOT sheetStackDischargeFaultCondition AND
   NOT sheetStackDischargeActive AND
   NOT sheetStackDischargePending THEN

    sheetStackDischargePending := TRUE;

    // EN: Clear current-cycle flags when a new cycle is accepted.
    sheetStackDischargeFault := FALSE;
    sheetStackDischargeFaultCode := 0;

    sheetStackDischargeCycleHasManualSkip := FALSE;
    sheetStackDischargeCycleHasTimeout := FALSE;

END_IF;


//==============================================================
// 7) Immediate abort condition
//==============================================================
// EN: Any relevant fault during an active/pending cycle aborts the
//     sequence and automatically returns to IDLE.
//     Loss of synchronized conveyor running also aborts the cycle.
abortCycle :=
    (
        sheetStackDischargeActive OR
        sheetStackDischargePending OR
        (sheetStackDischargeControlState <> E_SheetStackDischargeState.IDLE)
    )
    AND
    (
        sheetStackDischargeFaultCondition OR
        NOT synchronizedConveyorsRunning
    );


IF abortCycle THEN

    sheetStackDischargeConveyorRunRequest := FALSE;

    backstopTargetOverrideActive := FALSE;
    conveyorLevelerTargetOverrideActive := FALSE;

    sheetStackDischargePending := FALSE;
    sheetStackDischargeActive := FALSE;

    tonSheetStackDischarge(IN := FALSE);
    tonSheetStackDischargeStepTimeout(IN := FALSE);

    sheetStackDischargeFault := TRUE;

    sheetStackDischargeLastCycleOk := FALSE;
    sheetStackDischargeLastResultCode := 4;
    sheetStackDischargeLastFaultStepCode := sheetStackDischargeStateCode;
    sheetStackDischargeLastFaultCode := sheetStackDischargeFaultCode;

    sheetStackDischargeState := 'ABORTED';
    sheetStackDischargeStateCode := 90;

    // EN: Do not clear backstopManualInterventionActive here.
    //     If the cycle aborted before return, keeping the memory is safer
    //     for the next cycle.

    // EN: No latched FAULT state. Return to IDLE automatically.
    sheetStackDischargeControlState := E_SheetStackDischargeState.IDLE;


ELSE

    //==============================================================
    // 8) Sheet stack discharge state machine
    //==============================================================
    CASE sheetStackDischargeControlState OF

        E_SheetStackDischargeState.IDLE: // IDLE
            sheetStackDischargeState := 'IDLE';
            sheetStackDischargeStateCode := 0;

            sheetStackDischargeActive := FALSE;

            sheetStackDischargeConveyorRunRequest := FALSE;

            backstopTargetOverrideActive := FALSE;
            conveyorLevelerTargetOverrideActive := FALSE;

            tonSheetStackDischarge(IN := FALSE);
            tonSheetStackDischargeStepTimeout(IN := FALSE);

            IF sheetStackDischargePending THEN

                tonSheetStackDischarge(IN := FALSE);
                tonSheetStackDischargeStepTimeout(IN := FALSE);

                sheetStackDischargeControlState := E_SheetStackDischargeState.WAIT_SEPARATION;

            END_IF


        E_SheetStackDischargeState.WAIT_SEPARATION: // WAIT_SEPARATION
            sheetStackDischargeState := 'WAIT_SEPARATION';
            sheetStackDischargeStateCode := 5;

            sheetStackDischargeActive := FALSE;

            sheetStackDischargeConveyorRunRequest := FALSE;

            backstopTargetOverrideActive := FALSE;
            conveyorLevelerTargetOverrideActive := FALSE;

            tonSheetStackDischarge(IN := FALSE);

            // EN: Wait for conveyor speed control to finish sheet stack separation.
            tonSheetStackDischargeStepTimeout(
                IN := TRUE,
                PT := machineConfig.sheetStackDischargeWaitSeparationTimeout
            );

            IF sheetStackSeparationFinished THEN

                tonSheetStackDischargeStepTimeout(IN := FALSE);

                sheetStackDischargeControlState := E_SheetStackDischargeState.START_POSITIONING;


            ELSIF tonSheetStackDischargeStepTimeout.Q THEN

                // EN: Separation did not finish. Do not discharge.
                tonSheetStackDischargeStepTimeout(IN := FALSE);

                sheetStackDischargePending := FALSE;
                sheetStackDischargeActive := FALSE;

                sheetStackDischargeFault := TRUE;
                sheetStackDischargeFaultCode := 10;

                sheetStackDischargeLastCycleOk := FALSE;
                sheetStackDischargeLastResultCode := 3;
                sheetStackDischargeLastFaultStepCode := 5;
                sheetStackDischargeLastFaultCode := 10;

                sheetStackDischargeControlState := E_SheetStackDischargeState.IDLE;

            END_IF


        E_SheetStackDischargeState.START_POSITIONING: // START_DISCHARGE_POSITIONING
            sheetStackDischargeState := 'START_POSITIONING';
            sheetStackDischargeStateCode := 10;

            sheetStackDischargePending := FALSE;
            sheetStackDischargeActive := TRUE;
            sheetStackDischargeStarted := TRUE;

            tonSheetStackDischarge(IN := FALSE);
            tonSheetStackDischargeStepTimeout(IN := FALSE);

            //======================================================
            // EN: Latch programmed backstop target for this cycle.
            //     This is the normal position based on sheet length.
            //======================================================
            backstopProgrammedDischargeTargetMm :=
                LIMIT(
                    machineConfig.backstopMinPositionMm,
                    MAX(0.0, sheetLengthMm) +
                        machineConfig.backstopSheetLengthOffsetMm,
                    machineConfig.backstopMaxPositionMm
                );

            //======================================================
            // EN: Define safe opening base position.
            //
            // If the operator manually moved the backstop before the
            // automatic cycle, use the greater value between:
            // - programmed position
            // - last manual intervention position
            //
            // This prevents the automatic opening override from closing
            // the backstop onto the material.
            //
            // If there was no manual intervention, use only the programmed
            // position as the base.
            //======================================================
            IF backstopManualInterventionActive THEN

                backstopDischargeOpenBasePositionMm :=
                    MAX(
                        backstopProgrammedDischargeTargetMm,
                        backstopManualInterventionPositionMm
                    );

            ELSE

                backstopDischargeOpenBasePositionMm :=
                    backstopProgrammedDischargeTargetMm;

            END_IF;

            //======================================================
            // EN: Latch safe discharge open target.
            //     Offset is applied after selecting the safe base.
            //======================================================
            backstopDischargeOpenTargetMm :=
                LIMIT(
                    machineConfig.backstopMinPositionMm,
                    backstopDischargeOpenBasePositionMm +
                        machineConfig.backstopDischargeOpenOffsetMm,
                    machineConfig.backstopMaxPositionMm
                );

            // EN: Request safe backstop opening.
            //     Backstop control accepts it only in auto.
            backstopTargetOverrideActive := TRUE;
            backstopTargetOverridePositionMm := backstopDischargeOpenTargetMm;

            // EN: Request conveyor leveler to move up.
            //     The sequence does not wait for leveler feedback.
            conveyorLevelerTargetOverrideActive := TRUE;
            conveyorLevelerTargetOverridePositionMm :=
                machineConfig.conveyorLevelerMaxPositionMm;

            sheetStackDischargeControlState := E_SheetStackDischargeState.WAIT_BACKSTOP_POSITION;


        E_SheetStackDischargeState.WAIT_BACKSTOP_POSITION: // WAIT_BACKSTOP_POSITION
            sheetStackDischargeState := 'WAIT_BACKSTOP_POSITION';
            sheetStackDischargeStateCode := 20;

            sheetStackDischargeActive := TRUE;

            // EN: Keep safe latched backstop discharge target active.
            backstopTargetOverrideActive := TRUE;
            backstopTargetOverridePositionMm := backstopDischargeOpenTargetMm;

            // EN: Keep conveyor leveler up target active.
            //     Feedback is intentionally ignored for sequence progress.
            conveyorLevelerTargetOverrideActive := TRUE;
            conveyorLevelerTargetOverridePositionMm :=
                machineConfig.conveyorLevelerMaxPositionMm;

            // EN: If backstop is not in auto, do not wait for it.
            IF NOT backstopAutoCmd THEN

                sheetStackDischargeCycleHasManualSkip := TRUE;

                tonSheetStackDischargeStepTimeout(IN := FALSE);

                sheetStackDischargeControlState := E_SheetStackDischargeState.DISCHARGING;


            ELSIF backstopInPosition THEN

                tonSheetStackDischargeStepTimeout(IN := FALSE);

                sheetStackDischargeControlState := E_SheetStackDischargeState.DISCHARGING;


            ELSE

                tonSheetStackDischargeStepTimeout(
                    IN := TRUE,
                    PT := machineConfig.sheetStackDischargePositioningTimeout
                );

                IF tonSheetStackDischargeStepTimeout.Q THEN

                    // EN: Do not stay trapped waiting for backstop.
                    //     Continue the cycle, but record timeout diagnostic.
                    tonSheetStackDischargeStepTimeout(IN := FALSE);

                    sheetStackDischargeCycleHasTimeout := TRUE;

                    sheetStackDischargeFault := TRUE;
                    sheetStackDischargeFaultCode := 20;

                    sheetStackDischargeLastCycleOk := FALSE;
                    sheetStackDischargeLastResultCode := 3;
                    sheetStackDischargeLastFaultStepCode := 20;
                    sheetStackDischargeLastFaultCode := 20;

                    sheetStackDischargeControlState := E_SheetStackDischargeState.DISCHARGING;

                END_IF

            END_IF


        E_SheetStackDischargeState.DISCHARGING: // RUN_DISCHARGE_CONVEYOR
            sheetStackDischargeState := 'DISCHARGING';
            sheetStackDischargeStateCode := 30;

            sheetStackDischargeActive := TRUE;

            // EN: Keep safe latched backstop discharge target active
            //     while discharging.
            backstopTargetOverrideActive := TRUE;
            backstopTargetOverridePositionMm := backstopDischargeOpenTargetMm;

            // EN: Keep conveyor leveler up while discharging.
            conveyorLevelerTargetOverrideActive := TRUE;
            conveyorLevelerTargetOverridePositionMm :=
                machineConfig.conveyorLevelerMaxPositionMm;

            // EN: Request discharge conveyor run.
            //     Physical output is controlled by _SheetStackDischargeConveyorControl.
            sheetStackDischargeConveyorRunRequest := TRUE;

            // EN: If conveyor is not actually running, use start timeout.
            IF NOT sheetStackDischargeConveyorRun THEN

                tonSheetStackDischarge(IN := FALSE);

                tonSheetStackDischargeStepTimeout(
                    IN := TRUE,
                    PT := machineConfig.sheetStackDischargeConveyorStartTimeout
                );

                IF tonSheetStackDischargeStepTimeout.Q THEN

                    // EN: Conveyor did not start. Do not stay trapped.
                    tonSheetStackDischargeStepTimeout(IN := FALSE);

                    sheetStackDischargeConveyorRunRequest := FALSE;

                    sheetStackDischargeCycleHasTimeout := TRUE;

                    sheetStackDischargeFault := TRUE;
                    sheetStackDischargeFaultCode := 30;

                    sheetStackDischargeLastCycleOk := FALSE;
                    sheetStackDischargeLastResultCode := 3;
                    sheetStackDischargeLastFaultStepCode := 30;
                    sheetStackDischargeLastFaultCode := 30;

                    sheetStackDischargeControlState := E_SheetStackDischargeState.START_RETURN;

                END_IF


            ELSE

                // EN: Conveyor is running. Count real discharge time.
                tonSheetStackDischargeStepTimeout(IN := FALSE);

                tonSheetStackDischarge(
                    IN := TRUE,
                    PT := machineConfig.sheetStackDischargeTime
                );

                IF tonSheetStackDischarge.Q THEN

                    tonSheetStackDischarge(IN := FALSE);

                    sheetStackDischargeConveyorRunRequest := FALSE;

                    sheetStackDischargeControlState := E_SheetStackDischargeState.START_RETURN;

                END_IF

            END_IF


        E_SheetStackDischargeState.START_RETURN: // START_RETURN_POSITIONING
            sheetStackDischargeState := 'START_RETURN';
            sheetStackDischargeStateCode := 40;

            sheetStackDischargeActive := TRUE;

            sheetStackDischargeConveyorRunRequest := FALSE;

            tonSheetStackDischarge(IN := FALSE);
            tonSheetStackDischargeStepTimeout(IN := FALSE);

            // EN: Request backstop return to the latched programmed target.
            //     The override remains active until the backstop returns.
            backstopTargetOverrideActive := TRUE;
            backstopTargetOverridePositionMm :=
                backstopProgrammedDischargeTargetMm;

            // EN: Request conveyor leveler to return down.
            //     The sequence does not wait for leveler feedback.
            conveyorLevelerTargetOverrideActive := TRUE;
            conveyorLevelerTargetOverridePositionMm :=
                machineConfig.conveyorLevelerMinPositionMm;

            sheetStackDischargeControlState := E_SheetStackDischargeState.WAIT_BACKSTOP_RETURN;


        E_SheetStackDischargeState.WAIT_BACKSTOP_RETURN: // WAIT_BACKSTOP_RETURN
            sheetStackDischargeState := 'WAIT_BACKSTOP_RETURN';
            sheetStackDischargeStateCode := 50;

            sheetStackDischargeActive := TRUE;

            sheetStackDischargeConveyorRunRequest := FALSE;

            // EN: Keep backstop return target active.
            backstopTargetOverrideActive := TRUE;
            backstopTargetOverridePositionMm :=
                backstopProgrammedDischargeTargetMm;

            // EN: Keep conveyor leveler return target active.
            //     Feedback is intentionally ignored for sequence progress.
            conveyorLevelerTargetOverrideActive := TRUE;
            conveyorLevelerTargetOverridePositionMm :=
                machineConfig.conveyorLevelerMinPositionMm;

            // EN: If backstop is not in auto, do not wait for it.
            IF NOT backstopAutoCmd THEN

                sheetStackDischargeCycleHasManualSkip := TRUE;

                tonSheetStackDischargeStepTimeout(IN := FALSE);

                sheetStackDischargeControlState := E_SheetStackDischargeState.FINISH;


            ELSIF backstopInPosition THEN

                tonSheetStackDischargeStepTimeout(IN := FALSE);

                sheetStackDischargeControlState := E_SheetStackDischargeState.FINISH;


            ELSE

                tonSheetStackDischargeStepTimeout(
                    IN := TRUE,
                    PT := machineConfig.sheetStackDischargeReturnTimeout
                );

                IF tonSheetStackDischargeStepTimeout.Q THEN

                    // EN: Do not stay trapped waiting for return.
                    tonSheetStackDischargeStepTimeout(IN := FALSE);

                    sheetStackDischargeCycleHasTimeout := TRUE;

                    sheetStackDischargeFault := TRUE;
                    sheetStackDischargeFaultCode := 50;

                    sheetStackDischargeLastCycleOk := FALSE;
                    sheetStackDischargeLastResultCode := 3;
                    sheetStackDischargeLastFaultStepCode := 50;
                    sheetStackDischargeLastFaultCode := 50;

                    sheetStackDischargeControlState := E_SheetStackDischargeState.FINISH;

                END_IF

            END_IF


        E_SheetStackDischargeState.FINISH: // FINISH
            sheetStackDischargeState := 'FINISH';
            sheetStackDischargeStateCode := 60;

            sheetStackDischargeActive := FALSE;
            sheetStackDischargePending := FALSE;
            sheetStackDischargeFinished := TRUE;

            sheetStackDischargeConveyorRunRequest := FALSE;

            backstopTargetOverrideActive := FALSE;
            conveyorLevelerTargetOverrideActive := FALSE;

            tonSheetStackDischarge(IN := FALSE);
            tonSheetStackDischargeStepTimeout(IN := FALSE);

            IF sheetStackDischargeCycleHasTimeout THEN

                sheetStackDischargeLastCycleOk := FALSE;
                sheetStackDischargeLastResultCode := 3;

                // EN: Keep manual intervention memory after timeout.
                //     The backstop may not have returned correctly.

            ELSIF sheetStackDischargeCycleHasManualSkip THEN

                sheetStackDischargeLastCycleOk := FALSE;
                sheetStackDischargeLastResultCode := 2;
                sheetStackDischargeLastFaultStepCode := 0;
                sheetStackDischargeLastFaultCode := 0;

                sheetStackDischargeFault := FALSE;
                sheetStackDischargeFaultCode := 0;

                // EN: Keep manual intervention memory because the backstop
                //     was not controlled automatically.


            ELSE

                sheetStackDischargeLastCycleOk := TRUE;
                sheetStackDischargeLastResultCode := 1;
                sheetStackDischargeLastFaultStepCode := 0;
                sheetStackDischargeLastFaultCode := 0;

                sheetStackDischargeFault := FALSE;
                sheetStackDischargeFaultCode := 0;

                // EN: Cycle completed correctly and backstop returned to
                //     programmed target. Clear manual intervention memory.
                backstopManualInterventionActive := FALSE;
                backstopManualInterventionPositionMm := 0.0;

            END_IF

            // EN: Always return to IDLE automatically.
            sheetStackDischargeControlState := E_SheetStackDischargeState.IDLE;


    ELSE

        sheetStackDischargeControlState := E_SheetStackDischargeState.IDLE;

    END_CASE;

END_IF;
END_METHOD

//==============================================================
// SIMPLE STACKER — SHEET STACK DISCHARGE CONVEYOR CONTROL
// EN: Controls the sheet stack discharge conveyor.
//     Conveyor runs while manual button is pressed or while
//     automatic request is active and conveyor automatic mode is enabled.
//
// Fault code
// 0 = No fault
// 1 = Safety circuit not OK
// 2 = Discharge conveyor drive not OK
//==============================================================
METHOD _SheetStackDischargeConveyorControl
VAR
    manualRunRequest   : BOOL;
    automaticRunRequest: BOOL;
    finalRunRequest    : BOOL;
END_VAR
//==============================================================
// SIMPLE STACKER — SHEET STACK DISCHARGE CONVEYOR CONTROL
// EN: Controls the sheet stack discharge conveyor in manual pulse
//     or automatic sequence request.
//==============================================================


//==============================================================
// 1) Default outputs
//==============================================================
sheetStackDischargeConveyorRun := FALSE;
sheetStackDischargeConveyorSpeedRefMPM := 0.0;


//==============================================================
// 2) Run request selection
//==============================================================
// EN: Manual command is momentary. Conveyor runs while button is pressed.
manualRunRequest :=
    sheetStackDischargeConveyorManualRunCmd;


// EN: Automatic request is generated by the discharge sequence.
//     This conveyor is assumed to be available for automatic cycle
//     whenever the master system is enabled.
automaticRunRequest :=
    sheetStackDischargeConveyorRunRequest;


// EN: Master system enable blocks both manual and automatic movement.
finalRunRequest :=
    systemRunEnable AND
    (
        manualRunRequest OR
        automaticRunRequest OR
		backstopHomeRunning
    );


//==============================================================
// 3) Fault detection
//==============================================================
IF NOT safetyCircuitOk THEN

    sheetStackDischargeConveyorState := 'SAFETY_OFF';

    sheetStackDischargeConveyorFault := TRUE;
    sheetStackDischargeConveyorFaultCode := 1;


ELSIF NOT sheetStackDischargeConveyorDriveOk THEN

    sheetStackDischargeConveyorState := 'DRIVE_NOT_OK';

    sheetStackDischargeConveyorFault := TRUE;
    sheetStackDischargeConveyorFaultCode := 2;


ELSE

    //==============================================================
    // 4) Fault reset
    //==============================================================
    IF resetCmd THEN

        sheetStackDischargeConveyorFault := FALSE;
        sheetStackDischargeConveyorFaultCode := 0;

    END_IF;


    //==============================================================
    // 5) Conveyor output control
    //==============================================================
    IF sheetStackDischargeConveyorFault THEN

        sheetStackDischargeConveyorState := 'FAULT';

        sheetStackDischargeConveyorRun := FALSE;
        sheetStackDischargeConveyorSpeedRefMPM := 0.0;


    ELSIF NOT systemRunEnable THEN

        // EN: Master stop disables movement without generating a conveyor fault.
        sheetStackDischargeConveyorState := 'SYSTEM_DISABLED';

        sheetStackDischargeConveyorRun := FALSE;
        sheetStackDischargeConveyorSpeedRefMPM := 0.0;


    ELSIF finalRunRequest THEN

        IF automaticRunRequest THEN

            sheetStackDischargeConveyorState := 'AUTO_RUN';

        ELSE

            sheetStackDischargeConveyorState := 'MANUAL_RUN';

        END_IF;

        sheetStackDischargeConveyorRun := TRUE;

        sheetStackDischargeConveyorSpeedRefMPM :=
            LIMIT(
                0.0,
                machineConfig.sheetStackDischargeConveyorSpeedMPM,
                machineConfig.maximumSpeedMPM
            );


    ELSE

        sheetStackDischargeConveyorState := 'STOP';

        sheetStackDischargeConveyorRun := FALSE;
        sheetStackDischargeConveyorSpeedRefMPM := 0.0;

    END_IF

END_IF;
END_METHOD

//==============================================================
// SIMPLE STACKER — SYSTEM CONTROL
// EN: Master system run enable and automatic homing requests.
//==============================================================
METHOD _SystemControl

//==============================================================
// 1) Stop machine pulse on critical fault
//==============================================================
stopMachineFaultCondition :=
    NOT safetyCircuitOk OR
    NOT sheetConveyor1DriveOk OR
    NOT sheetConveyor2DriveOk OR
    NOT sheetConveyor3DriveOk OR
    NOT backstopDriveOk OR
    NOT conveyorLevelerDriveOk OR
    NOT sheetStackDischargeConveyorDriveOk;

rStopMachineFaultCondition :=
    stopMachineFaultCondition AND
    NOT stopMachineFaultConditionOld;

stopMachineFaultConditionOld :=
    stopMachineFaultCondition;

tpStopMachinePulse(
    IN := rStopMachineFaultCondition,
    PT := T#500MS
);

stopMachinePulse :=
    tpStopMachinePulse.Q;


//==============================================================
// 2) Default one-scan requests
//==============================================================
backstopAutoHomeRequest := FALSE;
conveyorLevelerAutoHomeRequest := FALSE;


//==============================================================
// 3) Master system run enable
//==============================================================
IF NOT safetyCircuitOk THEN

    systemRunEnable := FALSE;

ELSIF rStopCmd THEN

    systemRunEnable := FALSE;

ELSIF rStartCmd THEN

    systemRunEnable := TRUE;

END_IF;


//==============================================================
// 4) Automatic homing on system start
//==============================================================
// EN: Auto-home is generated only on the rising edge of startCmd.
//     Each axis must be enabled in automatic mode.
//     This prevents automatic movement of axes intentionally left in manual.
IF rStartCmd AND systemRunEnable THEN

    // Backstop auto-home
    IF backstopAutoCmd AND
       NOT backstopHomed AND
       NOT backstopFault THEN

        backstopAutoHomeRequest := TRUE;

    END_IF;


    // Conveyor leveler auto-home
    IF conveyorLevelerAutoCmd AND
       NOT conveyorLevelerHomed AND
       NOT conveyorLevelerFault THEN

        conveyorLevelerAutoHomeRequest := TRUE;

    END_IF;

END_IF;
END_METHOD

END_FUNCTION_BLOCK
